// Mitsubishi GX Works2 project: BookEX4_2 Ladder   PLC: Q13UDV

TYPE DateTime : STRUCT
  Year : INT;
  Month : INT;
  Day : INT;
  WeekDay : INT;
  iHour : INT;
  iMin : INT;
  iSec : INT;
  ms : INT;
END_STRUCT END_TYPE

TYPE Vector : STRUCT
  axisX : REAL;
  axisY : REAL;
  axisZ : REAL;
END_STRUCT END_TYPE

TYPE WordBit : STRUCT
  Data : DWORD;
  Flag : BOOL;
END_STRUCT END_TYPE

// global labels: Global
VAR_GLOBAL
  bVar0 AT M5000 : BOOL;
  abArray0 AT M5010 : ARRAY [0..49] OF BOOL;
  sStr0 AT D5000 : STRING[199];
  sStr1 AT D5100 : STRING[199];
  sStr2 AT D5200 : STRING[199];
  sStr3 AT D5300 : STRING[199];
  sStr4 AT D5400 : STRING[199];
  sStr5 AT D5500 : STRING[199];
  sStr6 AT D5600 : STRING[199];
  sStr7 AT D5700 : STRING[199];
  sStr8 AT D5800 : STRING[199];
  sStr9 AT D5900 : STRING[199];
  iVar0 AT D4500 : INT;
  iVar1 AT D4501 : INT;
  iVar2 AT D4502 : INT;
  iVar3 AT D4503 : INT;
  iVar4 AT D4504 : INT;
  iVar5 AT D4505 : INT;
  iVar6 AT D4506 : INT;
  iVar7 AT D4507 : INT;
  iVar8 AT D4508 : INT;
  iVar9 AT D4509 : INT;
  dVar0 AT D4510 : DINT;
  dVar1 AT D4512 : DINT;
  dVar2 AT D4514 : DINT;
  dVar3 AT D4516 : DINT;
  dVar4 AT D4518 : DINT;
  dVar5 AT D4520 : DINT;
  dVar6 AT D4522 : DINT;
  dVar7 AT D4524 : DINT;
  dVar8 AT D4526 : DINT;
  dVar9 AT D4528 : DINT;
  wVar0 AT D4530 : WORD;
  wVar1 AT D4531 : WORD;
  wVar2 AT D4532 : WORD;
  wVar3 AT D4533 : WORD;
  wVar4 AT D4534 : WORD;
  wVar5 AT D4535 : WORD;
  wVar6 AT D4536 : WORD;
  wVar7 AT D4537 : WORD;
  wVar8 AT D4538 : WORD;
  wVar9 AT D4539 : WORD;
  dwVar0 AT D4540 : DWORD;
  dwVar1 AT D4542 : DWORD;
  dwVar2 AT D4544 : DWORD;
  dwVar3 AT D4546 : DWORD;
  dwVar4 AT D4548 : DWORD;
  dwVar5 AT D4550 : DWORD;
  dwVar6 AT D4552 : DWORD;
  dwVar7 AT D4554 : DWORD;
  dwVar8 AT D4556 : DWORD;
  dwVar9 AT D4558 : DWORD;
  fsVar0 AT D4560 : REAL;
  fsVar1 AT D4562 : REAL;
  fsVar2 AT D4564 : REAL;
  fsVar3 AT D4566 : REAL;
  fsVar4 AT D4568 : REAL;
  fsVar5 AT D4570 : REAL;
  fsVar6 AT D4572 : REAL;
  fsVar7 AT D4574 : REAL;
  fsVar8 AT D4576 : REAL;
  fsVar9 AT D4578 : REAL;
  fdVar0 AT D4580 : LREAL;
  tTime0 AT D4620 : TIME;
  tTime1 AT D4622 : TIME;
  tTime2 AT D4624 : TIME;
  tTime3 AT D4626 : TIME;
  tTime4 AT D4628 : TIME;
  tTime5 AT D4630 : TIME;
  tTime6 AT D4632 : TIME;
  tTime7 AT D4634 : TIME;
  tTime8 AT D4636 : TIME;
  tTime9 AT D4638 : TIME;
  tTime10 AT D4640 : TIME;
  bVar1 AT M5001 : BOOL;
  bVar2 AT M5002 : BOOL;
  bVar3 AT M5003 : BOOL;
  bVar4 AT M5004 : BOOL;
  bVar5 AT M5005 : BOOL;
  bVar6 AT M5006 : BOOL;
  bVar7 AT M5007 : BOOL;
  bVar8 AT M5008 : BOOL;
  bVar9 AT M5009 : BOOL;
  abArray1 AT M5060 : ARRAY [0..49] OF BOOL;
  abArray2 AT M5110 : ARRAY [0..49] OF BOOL;
  abArray3 AT M5160 : ARRAY [0..49] OF BOOL;
  abArray4 AT M5210 : ARRAY [0..49] OF BOOL;
  abArray5 AT M5260 : ARRAY [0..49] OF BOOL;
  abArray6 AT M5310 : ARRAY [0..49] OF BOOL;
  abArray7 AT M5360 : ARRAY [0..49] OF BOOL;
  abArray8 AT M5410 : ARRAY [0..49] OF BOOL;
  abArray9 AT M5460 : ARRAY [0..49] OF BOOL;
  fdVar1 AT D4584 : LREAL;
  fdVar2 AT D4588 : LREAL;
  fdVar3 AT D4592 : LREAL;
  fdVar4 AT D4596 : LREAL;
  fdVar5 AT D4600 : LREAL;
  fdVar6 AT D4604 : LREAL;
  fdVar7 AT D4608 : LREAL;
  fdVar8 AT D4612 : LREAL;
  fdVar9 AT D4616 : LREAL;
  aSendData1 AT D100 : ARRAY [0..9] OF INT;
  aiTxData AT D4000 : ARRAY [0..99] OF INT;
  aiRxData AT D4100 : ARRAY [0..99] OF INT;
  iOpenOK AT D3900 : INT;
  iOpenERR AT D3901 : INT;
  iSendOK AT D3902 : INT;
  iSendERR AT D3903 : INT;
  iCloseOK AT D3906 : INT;
  iCloseERR AT D3907 : INT;
  iRecvOK AT D3904 : INT;
  iRecvERR AT D3905 : INT;
  aiTxData2 AT D4200 : ARRAY [0..99] OF INT;
  aiRxData2 AT D4300 : ARRAY [0..99] OF INT;
  iOpenOK2 AT D3908 : INT;
  iOpenERR2 AT D3909 : INT;
  iSendOK2 AT D3910 : INT;
  iSendERR2 AT D3911 : INT;
  iRecvOK2 AT D3912 : INT;
  iRecvERR2 AT D3913 : INT;
  iCloseOK2 AT D3914 : INT;
  iCloseERR2 AT D3915 : INT;
  iEOpenComp AT D3916 : INT;
  iEOpenReq AT D3917 : INT;
  iERecvFlag AT D3918 : INT;
  iOpenCode AT D3919 : INT;
  iSendCode AT D3920 : INT;
  iRecvCode AT D3921 : INT;
  iCloseCode AT D3922 : INT;
  iOpenCode2 AT D3923 : INT;
  iSendCode2 AT D3924 : INT;
  iRecvCode2 AT D3925 : INT;
  iCloseCode2 AT D3926 : INT;
  aRecvData1 AT D110 : ARRAY [0..9] OF INT;
  aSendData2 AT D120 : ARRAY [0..9] OF INT;
  aRecvData2 AT D130 : ARRAY [0..9] OF INT;
END_VAR
// user libraries (not included): HMI

PROGRAM ExLogic
VAR
  HMI05_1 : HMI05;
END_VAR
(* structured ladder/FBD written out as ST: instructions are called as NAME(EN, inputs, outputs); _pN, _eN, _tN stand for wires *)
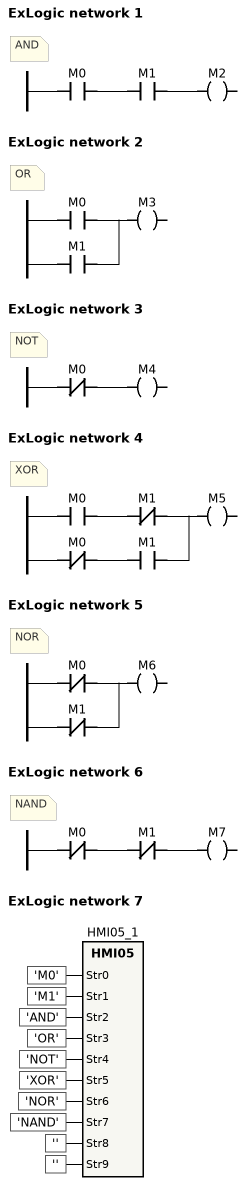
(* network 1 *)
(* AND *)
M2 := M0 AND M1;
(* network 2 *)
(* OR *)
M3 := M0 OR M1;
(* network 3 *)
(* NOT *)
M4 := NOT M0;
(* network 4 *)
(* XOR *)
M5 := (M0 AND NOT M1) OR (NOT M0 AND M1);
(* network 5 *)
(* NOR *)
M6 := (NOT M0) OR (NOT M1);
(* network 6 *)
(* NAND *)
M7 := NOT M0 AND NOT M1;
(* network 7 *)
HMI05_1(Str0 := 'M0', Str1 := 'M1', Str2 := 'AND', Str3 := 'OR', Str4 := 'NOT', Str5 := 'XOR', Str6 := 'NOR', Str7 := 'NAND', Str8 := '', Str9 := '');
END_PROGRAM

PROGRAM ExLogicFBD
VAR
  HMI05_1 : HMI05;
END_VAR
(* structured ladder/FBD written out as ST: instructions are called as NAME(EN, inputs, outputs); _pN, _eN, _tN stand for wires *)
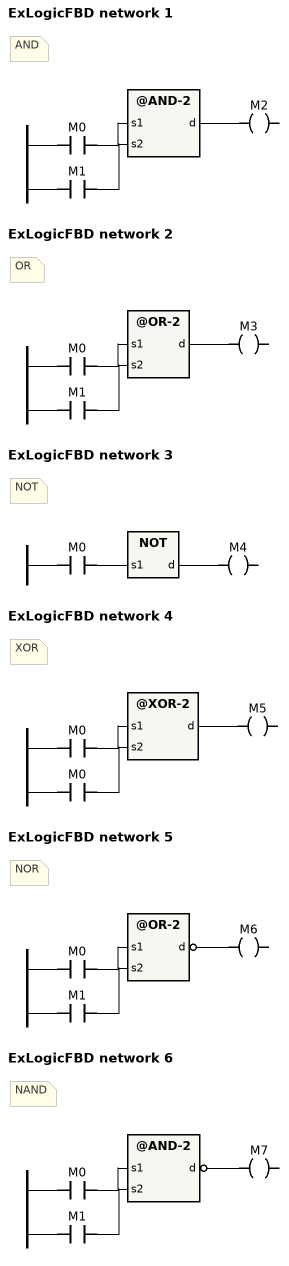
(* network 1 *)
(* AND *)
M2 := @AND-2(M0, M1);
(* network 2 *)
(* OR *)
M3 := @OR-2(M0, M1);
(* network 3 *)
(* NOT *)
M4 := NOT(M0);
(* network 4 *)
(* XOR *)
M5 := @XOR-2(M0, M0);
(* network 5 *)
(* NOR *)
M6 := NOT (@OR-2(M0, M1));
(* network 6 *)
(* NAND *)
M7 := NOT (@AND-2(M0, M1));
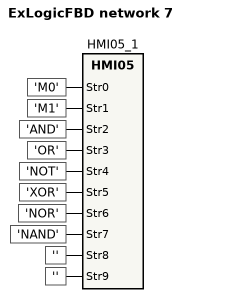
(* network 7 *)
HMI05_1(Str0 := 'M0', Str1 := 'M1', Str2 := 'AND', Str3 := 'OR', Str4 := 'NOT', Str5 := 'XOR', Str6 := 'NOR', Str7 := 'NAND', Str8 := '', Str9 := '');
END_PROGRAM

PROGRAM ExLatch
VAR
  HMI05_1 : HMI05;
END_VAR
(* structured ladder/FBD written out as ST: instructions are called as NAME(EN, inputs, outputs); _pN, _eN, _tN stand for wires *)
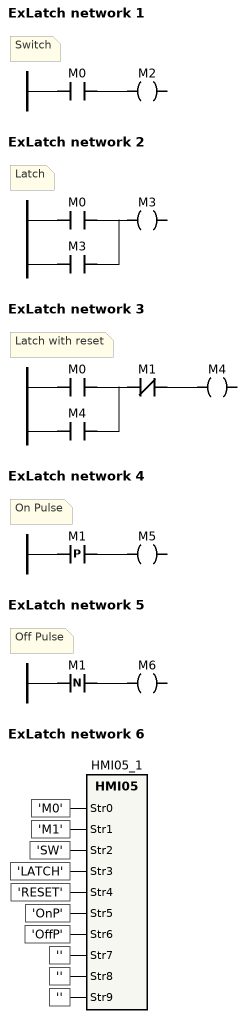
(* network 1 *)
(* Switch *)
M2 := M0;
(* network 2 *)
(* Latch *)
M3 := M0 OR M3;
(* network 3 *)
(* Latch with reset *)
M4 := (M0 OR M4) AND NOT M1;
(* network 4 *)
(* On Pulse *)
M5 := LDP(TRUE, M1);
(* network 5 *)
(* Off Pulse *)
M6 := LDF(TRUE, M1);
(* network 6 *)
HMI05_1(Str0 := 'M0', Str1 := 'M1', Str2 := 'SW', Str3 := 'LATCH', Str4 := 'RESET', Str5 := 'OnP', Str6 := 'OffP', Str7 := '', Str8 := '', Str9 := '');
END_PROGRAM

PROGRAM ExOnOff
VAR
  HMI05_1 : HMI05;
END_VAR
(* structured ladder/FBD written out as ST: instructions are called as NAME(EN, inputs, outputs); _pN, _eN, _tN stand for wires *)
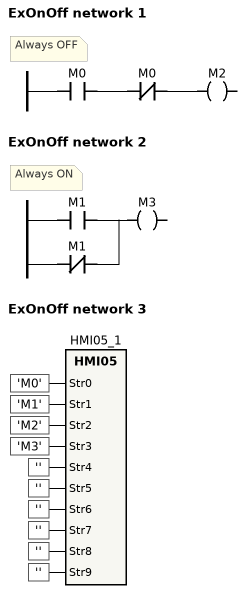
(* network 1 *)
(* Always OFF *)
M2 := M0 AND NOT M0;
(* network 2 *)
(* Always ON *)
M3 := M1 OR (NOT M1);
(* network 3 *)
HMI05_1(Str0 := 'M0', Str1 := 'M1', Str2 := 'M2', Str3 := 'M3', Str4 := '', Str5 := '', Str6 := '', Str7 := '', Str8 := '', Str9 := '');
END_PROGRAM

PROGRAM ExOSC
VAR
  TON_1 : TON;
  TON_2 : TON;
  HMI02_1 : HMI02;
END_VAR
(* structured ladder/FBD written out as ST: instructions are called as NAME(EN, inputs, outputs); _pN, _eN, _tN stand for wires *)
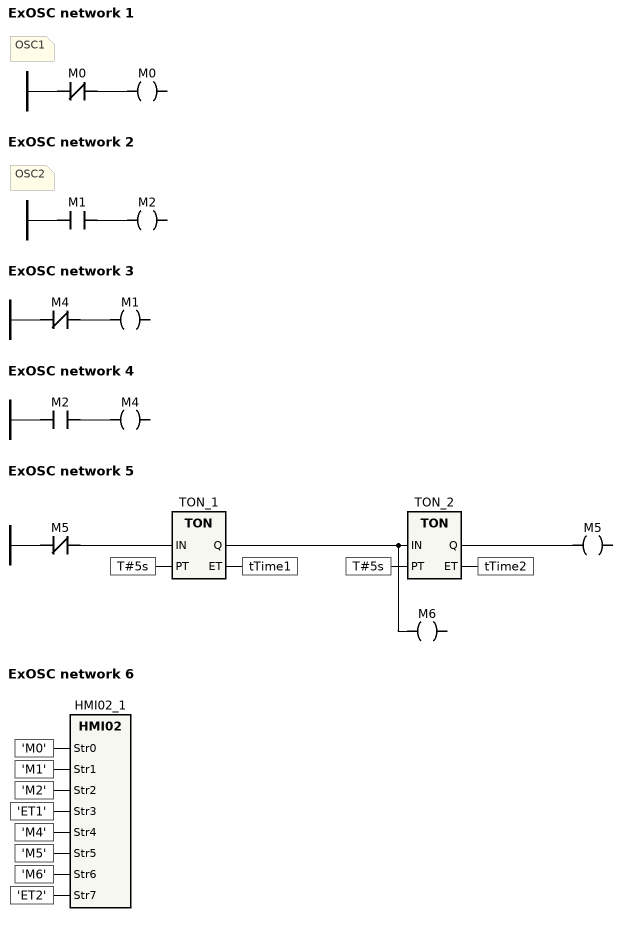
(* network 1 *)
(* OSC1 *)
M0 := NOT M0;
(* network 2 *)
(* OSC2 *)
M2 := M1;
(* network 3 *)
M1 := NOT M4;
(* network 4 *)
M4 := M2;
(* network 5 *)
TON_1(IN := NOT M5, PT := T#5s, ET => tTime1);
TON_2(IN := TON_1.Q, PT := T#5s, ET => tTime2);
M5 := TON_2.Q;
M6 := TON_1.Q;
(* network 6 *)
HMI02_1(Str0 := 'M0', Str1 := 'M1', Str2 := 'M2', Str3 := 'ET1', Str4 := 'M4', Str5 := 'M5', Str6 := 'M6', Str7 := 'ET2');
END_PROGRAM

PROGRAM ExInterlock
VAR
  HMI05_1 : HMI05;
END_VAR
(* structured ladder/FBD written out as ST: instructions are called as NAME(EN, inputs, outputs); _pN, _eN, _tN stand for wires *)
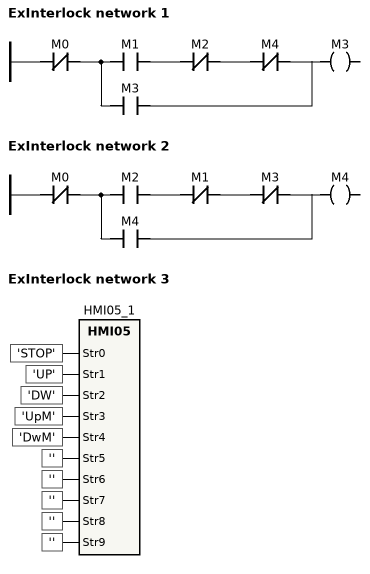
(* network 1 *)
_p1 := NOT M0;
M3 := (_p1 AND M1 AND NOT M2 AND NOT M4) OR (_p1 AND M3);
(* network 2 *)
_p1 := NOT M0;
M4 := (_p1 AND M2 AND NOT M1 AND NOT M3) OR (_p1 AND M4);
(* network 3 *)
HMI05_1(Str0 := 'STOP', Str1 := 'UP', Str2 := 'DW', Str3 := 'UpM', Str4 := 'DwM', Str5 := '', Str6 := '', Str7 := '', Str8 := '', Str9 := '');
END_PROGRAM

PROGRAM ExTFF
VAR
  HMI05_1 : HMI05;
END_VAR
(* structured ladder/FBD written out as ST: instructions are called as NAME(EN, inputs, outputs); _pN, _eN, _tN stand for wires *)
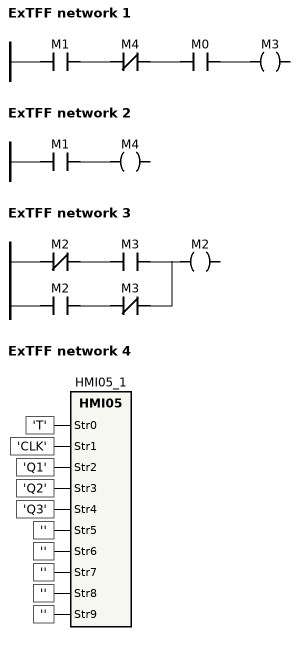
(* network 1 *)
M3 := M1 AND NOT M4 AND M0;
(* network 2 *)
M4 := M1;
(* network 3 *)
M2 := (NOT M2 AND M3) OR (M2 AND NOT M3);
(* network 4 *)
HMI05_1(Str0 := 'T', Str1 := 'CLK', Str2 := 'Q1', Str3 := 'Q2', Str4 := 'Q3', Str5 := '', Str6 := '', Str7 := '', Str8 := '', Str9 := '');
END_PROGRAM

PROGRAM ExDFF
VAR
  HMI05_1 : HMI05;
END_VAR
(* structured ladder/FBD written out as ST: instructions are called as NAME(EN, inputs, outputs); _pN, _eN, _tN stand for wires *)
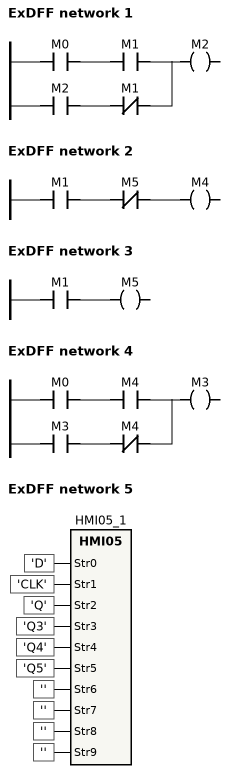
(* network 1 *)
M2 := (M0 AND M1) OR (M2 AND NOT M1);
(* network 2 *)
M4 := M1 AND NOT M5;
(* network 3 *)
M5 := M1;
(* network 4 *)
M3 := (M0 AND M4) OR (M3 AND NOT M4);
(* network 5 *)
HMI05_1(Str0 := 'D', Str1 := 'CLK', Str2 := 'Q', Str3 := 'Q3', Str4 := 'Q4', Str5 := 'Q5', Str6 := '', Str7 := '', Str8 := '', Str9 := '');
END_PROGRAM

PROGRAM ExJKFF
VAR
  HMI05_1 : HMI05;
END_VAR
(* structured ladder/FBD written out as ST: instructions are called as NAME(EN, inputs, outputs); _pN, _eN, _tN stand for wires *)
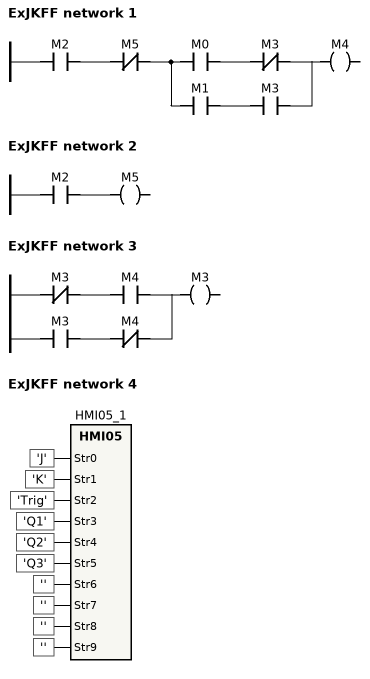
(* network 1 *)
_p1 := M2 AND NOT M5;
M4 := (_p1 AND M0 AND NOT M3) OR (_p1 AND M1 AND M3);
(* network 2 *)
M5 := M2;
(* network 3 *)
M3 := (NOT M3 AND M4) OR (M3 AND NOT M4);
(* network 4 *)
HMI05_1(Str0 := 'J', Str1 := 'K', Str2 := 'Trig', Str3 := 'Q1', Str4 := 'Q2', Str5 := 'Q3', Str6 := '', Str7 := '', Str8 := '', Str9 := '');
END_PROGRAM

PROGRAM ExTON
VAR
  TON_1 : TON;
  HMI03_1 : HMI03;
  TOF_1 : TOF;
END_VAR
(* structured ladder/FBD written out as ST: instructions are called as NAME(EN, inputs, outputs); _pN, _eN, _tN stand for wires *)
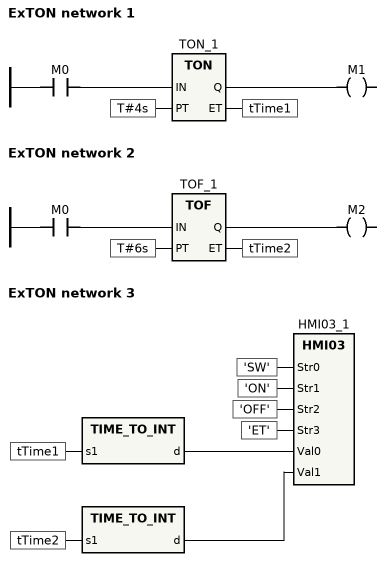
(* network 1 *)
TON_1(IN := M0, PT := T#4s, ET => tTime1);
M1 := TON_1.Q;
(* network 2 *)
TOF_1(IN := M0, PT := T#6s, ET => tTime2);
M2 := TOF_1.Q;
(* network 3 *)
HMI03_1(Str0 := 'SW', Str1 := 'ON', Str2 := 'OFF', Str3 := 'ET', Val0 := TIME_TO_INT(tTime1), Val1 := TIME_TO_INT(tTime2));
END_PROGRAM

PROGRAM ExTOF
VAR
  HMI03_1 : HMI03;
  TOF_1 : TOF;
END_VAR
(* structured ladder/FBD written out as ST: instructions are called as NAME(EN, inputs, outputs); _pN, _eN, _tN stand for wires *)
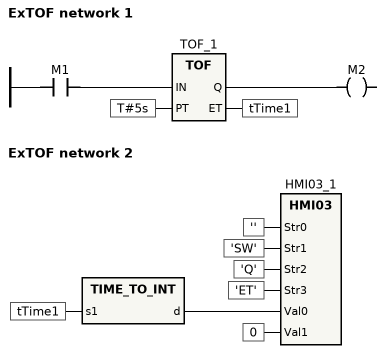
(* network 1 *)
TOF_1(IN := M1, PT := T#5s, ET => tTime1);
M2 := TOF_1.Q;
(* network 2 *)
HMI03_1(Str0 := '', Str1 := 'SW', Str2 := 'Q', Str3 := 'ET', Val0 := TIME_TO_INT(tTime1), Val1 := 0);
END_PROGRAM

PROGRAM EXTON_OFF
VAR
  TON_1 : TON;
  HMI03_1 : HMI03;
  TOF_1 : TOF;
END_VAR
(* structured ladder/FBD written out as ST: instructions are called as NAME(EN, inputs, outputs); _pN, _eN, _tN stand for wires *)
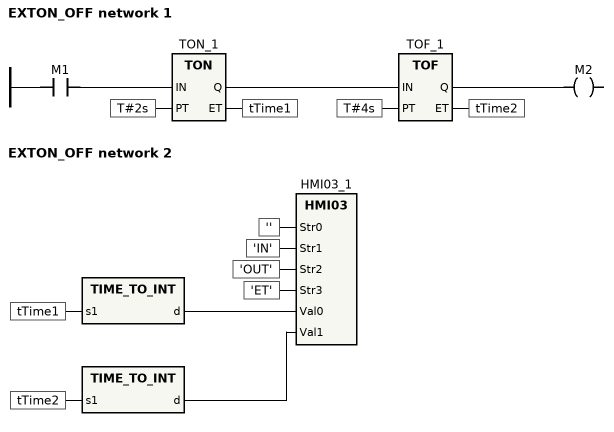
(* network 1 *)
TON_1(IN := M1, PT := T#2s, ET => tTime1);
TOF_1(IN := TON_1.Q, PT := T#4s, ET => tTime2);
M2 := TOF_1.Q;
(* network 2 *)
HMI03_1(Str0 := '', Str1 := 'IN', Str2 := 'OUT', Str3 := 'ET', Val0 := TIME_TO_INT(tTime1), Val1 := TIME_TO_INT(tTime2));
END_PROGRAM

PROGRAM ExMode
VAR
  swMan : BOOL;
  swSemi : BOOL;
  swAuto : BOOL;
  iMode : INT;
  HMI05_1 : HMI05;
END_VAR
(* structured ladder/FBD written out as ST: instructions are called as NAME(EN, inputs, outputs); _pN, _eN, _tN stand for wires *)
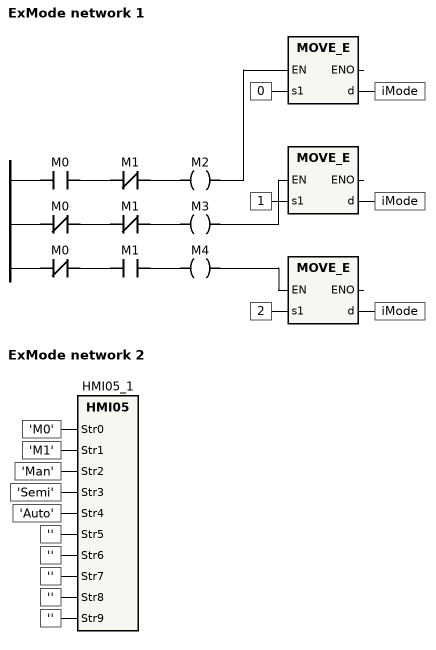
(* network 1 *)
_p1 := M0 AND NOT M1;
M2 := _p1;
MOVE_E(_p1, 0, iMode);
_p2 := NOT M0 AND NOT M1;
M3 := _p2;
MOVE_E(_p2, 1, iMode);
_p3 := NOT M0 AND M1;
M4 := _p3;
MOVE_E(_p3, 2, iMode);
(* network 2 *)
HMI05_1(Str0 := 'M0', Str1 := 'M1', Str2 := 'Man', Str3 := 'Semi', Str4 := 'Auto', Str5 := '', Str6 := '', Str7 := '', Str8 := '', Str9 := '');
END_PROGRAM
